Staubli VAL3: sendError.pgx

program sendError(num code, num argument)
  local num buffer[5]
begin
  buffer[0] = MAGIC_HEADER
  buffer[1] = 129
  buffer[2] = code

  toBinary(argument, 1, "2b", buffer[3])

  sioSet(socket, buffer)
end
